INTERFACE I_TestSuite

METHOD AddTest : BOOL
VAR_INPUT
    UnitTest : I_UnitTest;
END_VAR
END_METHOD

METHOD GetTest : I_UnitTest
VAR_INPUT
    Index : INT;
END_VAR
END_METHOD

PROPERTY Name : T_MaxString
GET
END_GET
END_PROPERTY

PROPERTY TestCount : INT
GET
END_GET
END_PROPERTY

END_INTERFACE

(* stored: Version 1.1.0.1, ProductVersion 3.1.4024.4
   Itf I_TestSuite: Id {80cf6ddf-a651-4ab2-891a-a7b3f91b2fb4}
   Method AddTest: Id {9c5890c3-cf8e-456f-a82e-905c99112e10}
   Method GetTest: Id {2dbfe228-23d5-4b93-863d-80e6ea34ac9f}
   Property Name: Id {5999c4b1-f0a0-4be0-877f-4919231e03ab}
   Get Get: Id {9d10175a-9fd1-4495-a9f8-024daded49b5}
   Property TestCount: Id {1bcfdb9f-9c31-4ab0-ad91-3c6f200fbb50}
   Get Get: Id {79276203-336f-4479-8b04-3a1f2d91fbed} *)
